{attribute 'qualified_only'}
VAR_GLOBAL
	
	MainPanel		:	SlitterMainOperatorPanel();//(StartPB, StopPB, StartLight, StopLight);

END_VAR

(* stored: Version 1.1.0.1, ProductVersion 3.1.4024.12
   GVL GVL: Id {2bccb817-fab3-47c8-906e-2d5f32b641f4} *)
